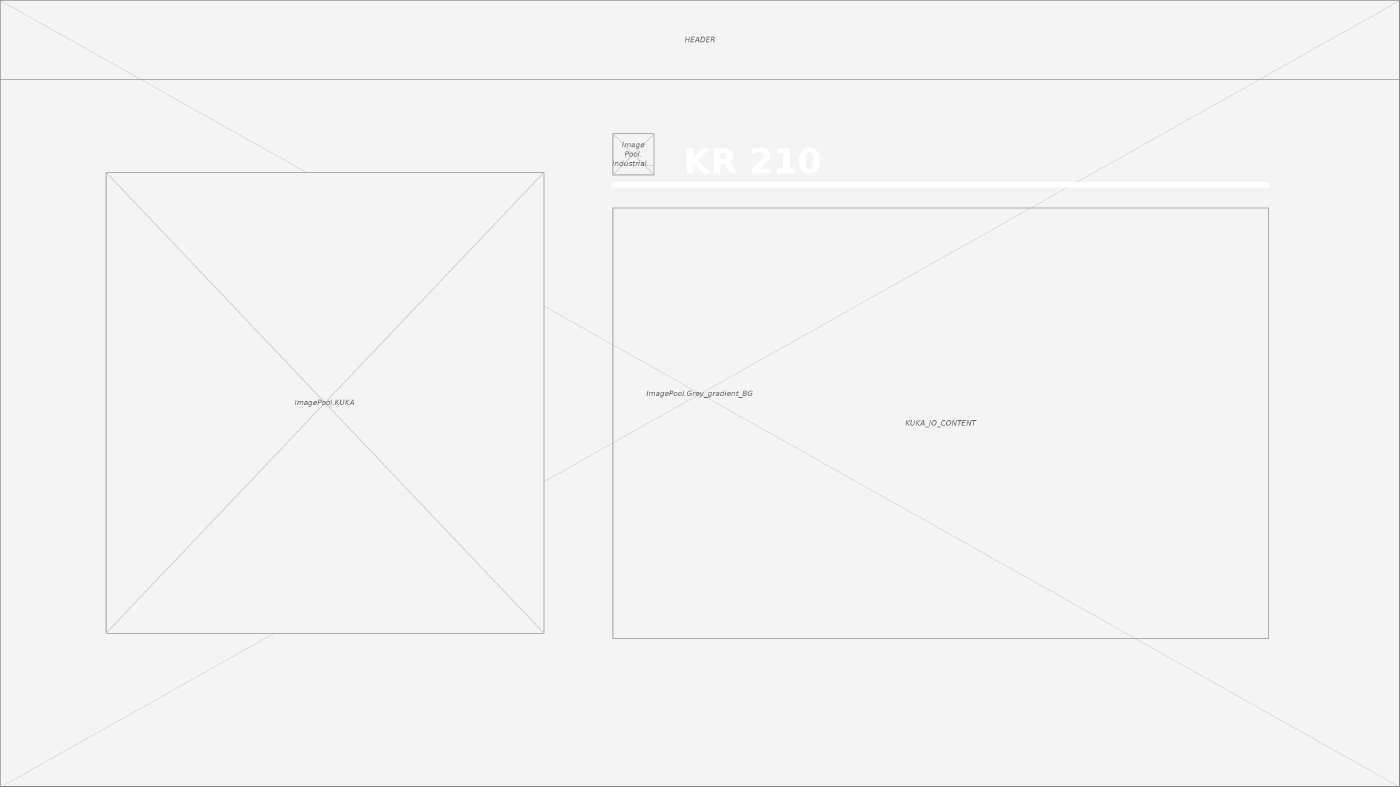
VISUALIZATION KUKA_PAGE  // 1920x1080
    Image (0,0 1920x1080), image: ImagePool.Grey_gradient_BG
    Rectangle (0,0 1920x1080)
    Image (145,236 601x633), image: ImagePool.KUKA
    Rectangle (885,184 294x74), "KR 210"
    Rectangle (840,250 900x7)
    Frame (0,0 1920x109)
        shows HEADER()
    TabControl (840,285 900x591)
        shows KUKA_IO_CONTENT()
        shows KUKA_PROG_CONTENT()
    Image (840,183 57x57), image: ImagePool.industrial-robot
END_VISUALIZATION

(* stored: Version 1.1.0.1, ProductVersion 3.1.4024.12
   Visu KUKA_PAGE: Id {95350db2-d5cc-43d5-8357-0c4e7ed32b56} *)
